# EPICS substitutions: dspamApp/Db/dspamCounter100.substitutions
file "dspamCounter.db" {
{N="\$(P)0"}
{N="\$(P)1"}
{N="\$(P)2"}
{N="\$(P)3"}
{N="\$(P)4"}
{N="\$(P)5"}
{N="\$(P)6"}
{N="\$(P)7"}
{N="\$(P)8"}
{N="\$(P)9"}
{N="\$(P)10"}
{N="\$(P)11"}
{N="\$(P)12"}
{N="\$(P)13"}
{N="\$(P)14"}
{N="\$(P)15"}
{N="\$(P)16"}
{N="\$(P)17"}
{N="\$(P)18"}
{N="\$(P)19"}
{N="\$(P)20"}
{N="\$(P)21"}
{N="\$(P)22"}
{N="\$(P)23"}
{N="\$(P)24"}
{N="\$(P)25"}
{N="\$(P)26"}
{N="\$(P)27"}
{N="\$(P)28"}
{N="\$(P)29"}
{N="\$(P)30"}
{N="\$(P)31"}
{N="\$(P)32"}
{N="\$(P)33"}
{N="\$(P)34"}
{N="\$(P)35"}
{N="\$(P)36"}
{N="\$(P)37"}
{N="\$(P)38"}
{N="\$(P)39"}
{N="\$(P)40"}
{N="\$(P)41"}
{N="\$(P)42"}
{N="\$(P)43"}
{N="\$(P)44"}
{N="\$(P)45"}
{N="\$(P)46"}
{N="\$(P)47"}
{N="\$(P)48"}
{N="\$(P)49"}
{N="\$(P)50"}
{N="\$(P)51"}
{N="\$(P)52"}
{N="\$(P)53"}
{N="\$(P)54"}
{N="\$(P)55"}
{N="\$(P)56"}
{N="\$(P)57"}
{N="\$(P)58"}
{N="\$(P)59"}
{N="\$(P)60"}
{N="\$(P)61"}
{N="\$(P)62"}
{N="\$(P)63"}
{N="\$(P)64"}
{N="\$(P)65"}
{N="\$(P)66"}
{N="\$(P)67"}
{N="\$(P)68"}
{N="\$(P)69"}
{N="\$(P)70"}
{N="\$(P)71"}
{N="\$(P)72"}
{N="\$(P)73"}
{N="\$(P)74"}
{N="\$(P)75"}
{N="\$(P)76"}
{N="\$(P)77"}
{N="\$(P)78"}
{N="\$(P)79"}
{N="\$(P)80"}
{N="\$(P)81"}
{N="\$(P)82"}
{N="\$(P)83"}
{N="\$(P)84"}
{N="\$(P)85"}
{N="\$(P)86"}
{N="\$(P)87"}
{N="\$(P)88"}
{N="\$(P)89"}
{N="\$(P)90"}
{N="\$(P)91"}
{N="\$(P)92"}
{N="\$(P)93"}
{N="\$(P)94"}
{N="\$(P)95"}
{N="\$(P)96"}
{N="\$(P)97"}
{N="\$(P)98"}
{N="\$(P)99"}
}
